Fanuc KAREL source: ko00035.KL

-- PROVISIONAL review KL for V770-1; original PC SHA256 fad0f60b1e7a7723099e2321f113b8ee2d0ff3104697dad36bf8df52c37cb53a
-- Incomplete behavior may be omitted. Consult companion uncertainty JSON. Do not deploy.
PROGRAM KO00035
%NOLOCKGROUP
BEGIN
  -- UNRESOLVED_PC offsets 5-12; opcodes 9D,23
  -- UNRESOLVED_PC offsets 17-66; opcodes 27,27,49,7E,AD,22,1C,22,31,7E,4A
  -- UNRESOLVED_PC offsets 71-75; opcodes 7F
END KO00035
